// LS Electric XG5000 project: test1
// PLC NewPLC
// module base 0 slot 0: 입출력 모듈:XBC-DR20S (DC 24V 입력 12점, 릴레이 출력 8점)

PROGRAM NewProgram (task: 스캔 프로그램)

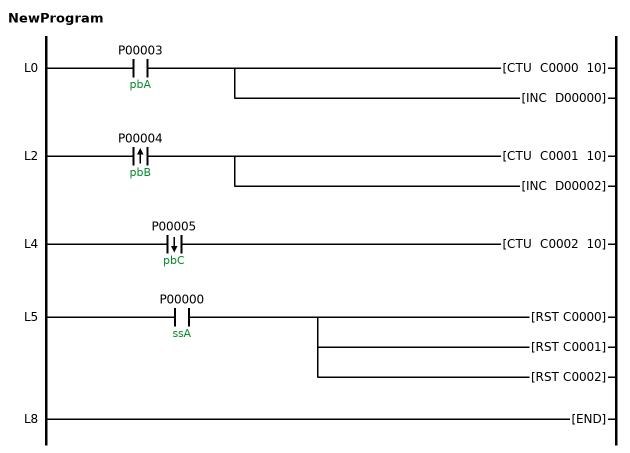
; L0
LOAD      P00003	// pbA
CTU       C0000 10
INC       D00000
; L2
LOADP     P00004	// pbB
CTU       C0001 10
INC       D00002
; L4
LOADN     P00005	// pbC
CTU       C0002 10
; L5
LOAD      P00000	// ssA
RST       C0000
RST       C0001
RST       C0002
; L8
END

VARIABLES AND COMMENTS (devices not used above)
P00040	BIT	plA
P00041	BIT	plB
P00042	BIT	plC
P00043	BIT	plD
P00044	BIT	plE
P00001	BIT	ssB
P00002	BIT	ssC